{attribute 'GeneratedUsingTerminal: EK1122-0000-0018'}
{attribute addProperty BoxType "EK1122-0000-0018"}
{attribute addProperty Id "Beckhoff_ER6xxxsub_EK1100EK1100_1FC0878B2A_0001_ER6001_0002_0016ER6001_40883D0360A_0002_ER6001_0002_0021ER6001_40883D0360A_0003_ER6002_0002_0021ER6002_7F53816A108A_0004_ER6002_0002_0022ER6002_7BE6B617108A_0005_ER6002_0002_0023ER6002_7BE6B617108"}
{attribute addProperty CRC "3176207089"}
{attribute addProperty Size "446"}
TYPE Beckhoff_ER6xxxEK1122_BD5112F1 EXTENDS EK1122_1FC0878B :
STRUCT
	{attribute addProperty Name "Beckhoff ER6xxxsub EK1100"}
	{attribute addProperty PreviousPort "Beckhoff ER6xxxEK1122 : D"}
	Beckhoff_ER6xxxsub_EK1100 : EK1100_1FC0878B;
	{attribute addProperty Name "A_0001(ER6001-0002-0016)"}
	{attribute addProperty PreviousPort "Beckhoff ER6xxxsub EK1100 : C"}
	A_0001_ER6001_0002_0016 : ER6001_40883D03;
	{attribute addProperty Name "A_0002(ER6001-0002-0021)"}
	{attribute addProperty PreviousPort "A_0001(ER6001-0002-0016) : B"}
	A_0002_ER6001_0002_0021 : ER6001_40883D03;
	{attribute addProperty Name "A_0003(ER6002-0002-0021)"}
	{attribute addProperty PreviousPort "A_0002(ER6001-0002-0021) : B"}
	A_0003_ER6002_0002_0021 : ER6002_7F53816A;
	{attribute addProperty Name "A_0004(ER6002-0002-0022)"}
	{attribute addProperty PreviousPort "A_0003(ER6002-0002-0021) : B"}
	A_0004_ER6002_0002_0022 : ER6002_7BE6B617;
	{attribute addProperty Name "A_0005(ER6002-0002-0023)"}
	{attribute addProperty PreviousPort "A_0004(ER6002-0002-0022) : B"}
	A_0005_ER6002_0002_0023 : ER6002_7BE6B617;
END_STRUCT
END_TYPE

(* stored: Version 1.2.0.0, ProductVersion 3.1.4024.9
   DUT Beckhoff_ER6xxxEK1122_BD5112F1: Id {8179b033-9e7e-4658-b102-4caedda26b6d} *)
